FUNCTION_BLOCK FB_Pid
VAR
END_VAR

END_FUNCTION_BLOCK

(* stored: Version 1.1.0.1
   POU FB_Pid: Id {87deac38-ac60-467f-aaaf-cdf4d170d96b}, SpecialFunc None *)
